TYPE ST_WaferTransferResponse :
STRUCT
	// Non-zero and unique within one Module; array index is storage only.
	EndpointId : UDINT;
	WaferHandlingType : E_WaferHandlingType;
	Capability : E_TransferCapability;

	Send : ST_WaferTransferStatus;
	Receive : ST_WaferTransferStatus;

	// Passive only
	SendReady : BOOL;
	ReceiveReady : BOOL;

	//TransferState : E_TransferState;
END_STRUCT
END_TYPE

(* stored: Version 1.1.0.1, ProductVersion 3.1.4026.18
   DUT ST_WaferTransferResponse: Id {14f9d5f9-39d1-4854-bedd-e4f7b43e695c} *)
